TYPE T_JXCE1_AccDec : REAL; END_TYPE

(* stored: Version 1.1.0.1, ProductVersion 3.1.4024.15
   DUT T_JXCE1_AccDec: Id {991537b8-fe56-0d3e-05dc-4f0129b0f89e} *)
